PROGRAM MAIN_1
VAR
	myAxisA : FB_Axis;
	myAxisB : FB_Axis;
	myAxisVirtual : FB_Axis;
	myAxisStepper : FB_Axis;
	fbAxisStMachine : FB_AxisStMachine;
END_VAR

//myAxisA(AxisInOut := GVL.Axis_servoA);
//myAxisB(AxisInOut := GVL.Axis_servoB);
//myAxisVirtual(AxisInOut := GVL.Axis_servoVirtual);
//myAxisStepper(AxisInOut := GVL.Axis_servo);
//fbAxisStMachine(AxisInOut := GVL.Axis_servoA);

END_PROGRAM

(* stored: Version 1.1.0.1, ProductVersion 3.1.4024.12
   POU MAIN_1: Id {820171f7-8670-42df-9df1-221fdd638619}, SpecialFunc None *)
